Yaskawa INFORM job: R1_S1_MAIN.JBI

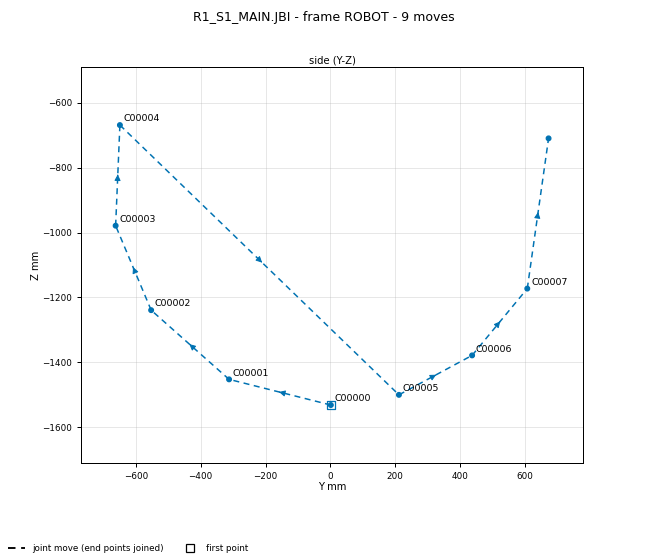
[picture p0: tool path of R1_S1_MAIN.JBI in frame ROBOT, 9 of 9 moves have a stored position in this frame; points joined in program order, loops and branches not executed]
/JOB
//NAME R1_S1_MAIN
///FOLDERNAME INNE
//POS
///NPOS 9,9,0,0,0,0
///TOOL 0
///POSTYPE ROBOT
///RECTAN
///RCONF 0,0,0,0,0,0,0,0,0,0,0,0,0,0,0,0,0,0,0,0,0,0,0,0
C00000=1534.930,1.471,-1531.968,-2.1356,-0.0600,-32.5919
C00001=1533.634,-312.442,-1452.824,-24.5055,-13.7608,-29.8326
C00002=1532.741,-552.767,-1239.427,-51.0575,-25.7855,-20.6576
C00003=1532.195,-662.301,-978.833,-76.0715,-31.5725,-8.4886
C00004=1532.211,-649.151,-668.546,-107.8786,-31.5734,8.4831
C00005=1535.036,211.475,-1500.581,12.9254,5.5860,-25.6716
C00006=1535.473,437.164,-1378.891,36.3236,15.7221,-21.2729
C00007=1536.159,607.368,-1172.890,56.0404,21.8735,-14.8552
C00008=1536.353,673.008,-709.551,98.0612,26.0824,2.8967
BC00000=1.074,829.375,857.934
BC00001=1.074,829.369,857.929
BC00002=1.074,829.369,857.929
BC00003=1.074,829.369,857.929
BC00004=1.074,829.369,857.929
BC00005=1.074,829.369,857.925
BC00006=1.074,829.369,857.925
BC00007=1.074,829.369,857.925
BC00008=1.074,829.369,857.925
//INST
///DATE 2023/10/04 15:16
///ATTR SC,RW,RJ
////FRAME ROBOT
///GROUP1 RB1,BS1
NOP
MOVJ C00000 BC00000 VJ=0.78
MOVJ C00001 BC00001 VJ=0.78
MOVJ C00002 BC00002 VJ=0.78
MOVJ C00003 BC00003 VJ=0.78
MOVJ C00004 BC00004 VJ=0.78
MOVJ C00005 BC00005 VJ=0.78
MOVJ C00006 BC00006 VJ=0.78
MOVJ C00007 BC00007 VJ=0.78
MOVJ C00008 BC00008 VJ=0.78
END
